PROGRAM Main_Batch
VAR
	FB_Tank_1 : FB_Tank;
END_VAR

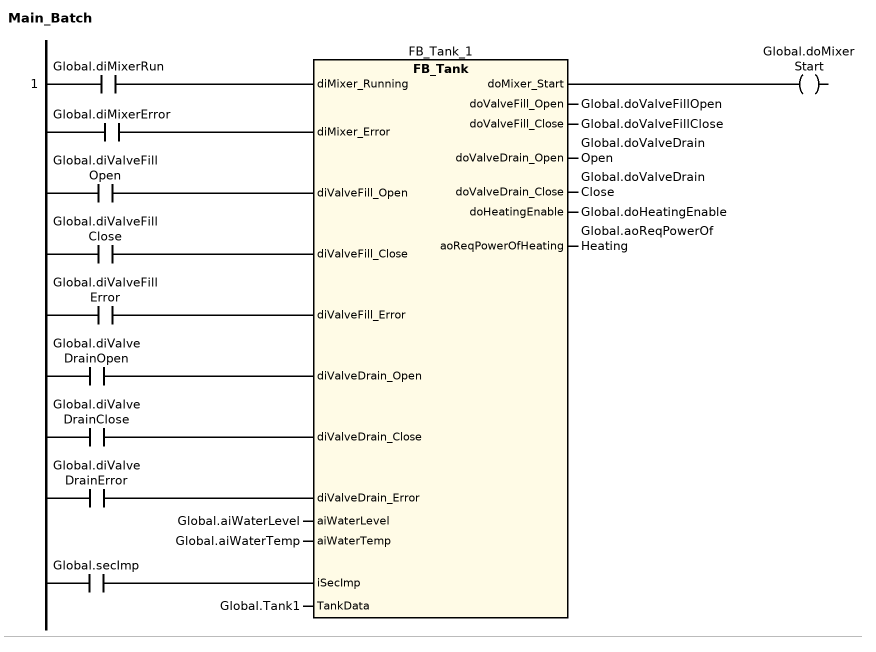
// NETWORK 1
FB_Tank_1(
    diMixer_Running := Global.diMixerRun,
    diMixer_Error := Global.diMixerError,
    diValveFill_Open := Global.diValveFillOpen,
    diValveFill_Close := Global.diValveFillClose,
    diValveFill_Error := Global.diValveFillError,
    diValveDrain_Open := Global.diValveDrainOpen,
    diValveDrain_Close := Global.diValveDrainClose,
    diValveDrain_Error := Global.diValveDrainError,
    aiWaterLevel := Global.aiWaterLevel,
    aiWaterTemp := Global.aiWaterTemp,
    iSecImp := Global.secImp,
    TankData := Global.Tank1,
    doValveFill_Open => Global.doValveFillOpen,
    doValveFill_Close => Global.doValveFillClose,
    doValveDrain_Open => Global.doValveDrainOpen,
    doValveDrain_Close => Global.doValveDrainClose,
    doHeatingEnable => Global.doHeatingEnable,
    aoReqPowerOfHeating => Global.aoReqPowerOfHeating); // FB_Tank
Global.doMixerStart := FB_Tank_1.doMixer_Start;

END_PROGRAM

(* stored: Version 1.1.0.1, ProductVersion 3.1.4024.13
   POU Main_Batch: Id {719b888b-042e-4776-9f4f-d0959c3a537e}, SpecialFunc None *)
